(* CODESYS project Test_Modbus_HMI.project
   Title: Test_Modbus_TCP_IP
   Version: 0.0.0.0
   Author: serbogr1

Project tree, tasks and I/O mapping:
  MyController : TM241CE40R, Schneider Electric, order no. TM241CE40R, version 4.0.6.18
    application Application
      task MAST (cyclic, interval 20 ms, priority 15, watchdog 100 ms x 1) calls Cilindros
      global variables GVL
      program MyPOU [ST]
      visualisation ModbusTCP
      program Cilindros [LD]
    DI : Digital Inputs, Schneider Electric, version 4.0.6.18
        input  idwDI_IDW0 : DWORD  // IDW0
        input  ibDI_IB1 : BYTE  // IB1
    DQ : Digital Outputs, Schneider Electric, version 4.0.6.18
        output qwDQ_QW0 : WORD  // QW0
        output qbDQ_QB1 : BYTE  // QB1
    Counters : Counters, Schneider Electric, version 4.0.6.18
    Pulse_Generators : Pulse Generators, Schneider Electric, version 4.0.6.18
    Cartridge_1 : Cartridge, Schneider Electric, version 4.0.6.18
    Cartridge_2 : Cartridge, Schneider Electric, version 4.0.6.18
    IO_Bus : IO bus - TM3, Schneider Electric, version 4.0.6.18
    COM_Bus : COM bus, Schneider Electric, version 4.0.6.18
    Ethernet_1 : Ethernet Network, Schneider Electric, version 4.0.6.18
        settings: IPAddress = [172, 16, 191, 108]; SubnetMask = [255, 255, 255, 0]; GatewayAddress = [172, 16, 191, 1]; WebServer = TRUE; FTP Server = TRUE; SoMachine Protocol = TRUE; Modbus Server = TRUE; NetManage Protocol = TRUE; SNMP protocol = TRUE; Enable Routing = FALSE; WebVisu protocol = TRUE; DHCP Server Active = FALSE
    Serial_Line_1 : Serial line, Schneider Electric, version 4.0.6.18
    Serial_Line_2 : Serial line, Schneider Electric, version 4.0.6.18
  text list GlobalTextList
*)

// MyController/Application/GVL
VAR_GLOBAL
END_VAR

// MyController/Application/Cilindros
PROGRAM Cilindros
VAR
	Sacar_CSuperior AT %QX0.4: BOOL;
	Boton_CSuperior AT %MX0.0: BOOL;
	Boton_CCentral AT %MX0.1: BOOL;
	Sacar_CCentral AT %QX0.5: BOOL;
	Boton_CInferior AT %MX0.2: BOOL;
	Sacar_CInferior AT %QX0.7: BOOL;
	Boton_MCCentral AT %MX0.3: BOOL;
	Boton_MCInferior AT %MX0.4: BOOL;
	Meter_CCentral AT %QX0.6: BOOL;
	Ventosa AT %QX1.3: BOOL;
	Boton_Ventosa AT %MX0.5: BOOL;
	Boton_Abrir_Pinza AT %MX0.7: BOOL;
	Boton_Cerrar_Pinza AT %MX0.6: BOOL;
	Abrir_Pinza AT %QX1.1: BOOL;
	Cerrar_Pinza AT %QX1.0: BOOL;
END_VAR

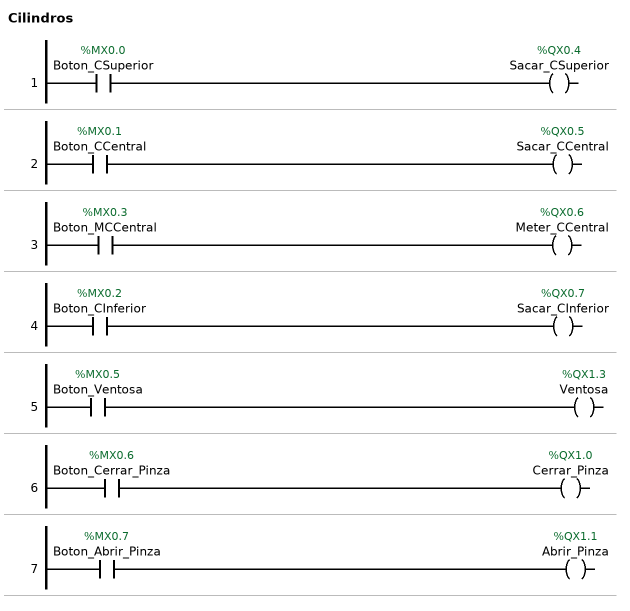
// NETWORK 1
//   Boton_CSuperior: AT %MX0.0
//   Sacar_CSuperior: AT %QX0.4
Sacar_CSuperior := Boton_CSuperior;

// NETWORK 2
//   Boton_CCentral: AT %MX0.1
//   Sacar_CCentral: AT %QX0.5
Sacar_CCentral := Boton_CCentral;

// NETWORK 3
//   Boton_MCCentral: AT %MX0.3
//   Meter_CCentral: AT %QX0.6
Meter_CCentral := Boton_MCCentral;

// NETWORK 4
//   Boton_CInferior: AT %MX0.2
//   Sacar_CInferior: AT %QX0.7
Sacar_CInferior := Boton_CInferior;

// NETWORK 5
//   Boton_Ventosa: AT %MX0.5
//   Ventosa: AT %QX1.3
Ventosa := Boton_Ventosa;

// NETWORK 6
//   Boton_Cerrar_Pinza: AT %MX0.6
//   Cerrar_Pinza: AT %QX1.0
Cerrar_Pinza := Boton_Cerrar_Pinza;

// NETWORK 7
//   Boton_Abrir_Pinza: AT %MX0.7
//   Abrir_Pinza: AT %QX1.1
Abrir_Pinza := Boton_Abrir_Pinza;

END_PROGRAM

// MyController/Application/MyPOU
PROGRAM MyPOU
VAR
	HMI_INPUT AT %MW100: WORD;
	HIMI_OUTPUT AT %MW110: WORD;
END_VAR

END_PROGRAM

// MyController/Application/ModbusTCP
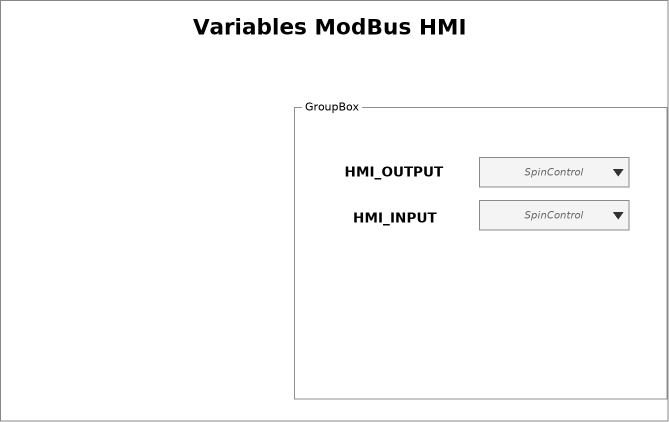
VISUALIZATION ModbusTCP  // 669x422
    Label (150,12 360x30), "Variables ModBus HMI"
    Label (57,115 150x30)
    GroupBox (294,99 373x300), "GroupBox"
        Label (25,58 150x30), "HMI_OUTPUT"
        Label (26,104 150x30), "HMI_INPUT"
        SpinControl (185,58 150x30), variable: MyPOU.HIMI_OUTPUT
        SpinControl (185,101 150x30), variable: MyPOU.HMI_INPUT
        Label (30,197 150x30)
        Label (31,245 150x30)
        Label (32,291 150x30)
END_VISUALIZATION
